{attribute addProperty BoxType "AT2020-0250-0019"}
{attribute addProperty Id "StatusAT %I*UINT1621Current_actual_value_ChAT %I*ARRAY[0 ..14] OF INT240300"}
{attribute addProperty CRC "1710915245"}
{attribute addProperty SizeInBites "256"}
{attribute addProperty SizeInBytes "32"}
TYPE CC_Inputs_9818D8D8 :
STRUCT
	{attribute addProperty Name "Status"}
	Status AT %I* : UINT;
	{attribute addProperty Name "Current_actual_value_Ch"}
	Current_actual_value_Ch AT %I* : ARRAY[0 ..14] OF INT;
END_STRUCT
END_TYPE

(* stored: Version 1.2.0.0, ProductVersion 3.1.4024.9
   DUT CC_Inputs_9818D8D8: Id {cfe20f0d-f945-4133-939b-168b0d6e04aa} *)
